// TIA Portal V20 export
TYPE "LWONIK_typeSafetyZoneManualEnable"
// stored: Access Published
   STRUCT
      SafetyZone1OpManualOn : Bool;   // SafetyZone1_PHMI Enable / HMI Enable On
      SafetyZone2OpManualOn : Bool;   // SafetyZone2_PHMI Enable / HMI Enable On
      SafetyZone3OpManualOn : Bool;   // SafetyZone3_PHMI Enable / HMI Enable On
      SafetyZone4OpManualOn : Bool;   // SafetyZone4_PHMI Enable / HMI Enable On
      SafetyZone5OpManualOn : Bool;   // SafetyZone5_PHMI Enable / HMI Enable On
   END_STRUCT;
END_TYPE
